// TIA Portal V19 export
VAR_GLOBAL   // PLC tag table "Safety_IO"
   IS_ZAxisBrakeFeedback AT %I500.0 : Bool;   // Robot Z axis brake status feedback channel 1   {ExternalAccessible false}
   IS_ZAxisBrakeFeedback_Ch2 AT %I500.4 : Bool;   // Robot Z axis brake status feedback channel 2   {ExternalAccessible false}
   OS_OpenZAxisBrake AT %Q508.0 : Bool;   // Open Z axis brake   {ExternalAccessible false}
   ISS_OpenZAxisBrake AT %I508.0 : Bool;   // State Open Z axis brake   {ExternalAccessible false}
   ISS_ZAxisBrakeFeedback AT %I501.0 : Bool;   // State Robot Z axis brake status feedback channel 1   {ExternalAccessible false}
   ISS_ZAxisBrakeFeedback_Ch2 AT %I501.4 : Bool;   // State Robot Z axis brake status feedback channel 2   {ExternalAccessible false}
   IS_AutomaticMode AT %I514.0 : Bool;   // True if Automatic mode is selected.   {ExternalAccessible false}
   IS_DriveEnableFeedback AT %I514.1 : Bool;   // True if the power to the motors is enabled.   {ExternalAccessible false}
   IS_EnableSwitch AT %I514.2 : Bool;   // True when the enable switch is activated   {ExternalAccessible false}
   IS_LocalEStopStatus AT %I514.3 : Bool;   // False if the emergency stop on the FlexPendant is pressed.   {ExternalAccessible false}
   IS_ManualFullSpeedMode AT %I514.4 : Bool;   // True if manual full speed mode is selected.   {ExternalAccessible false}
   IS_ManualMode AT %I514.5 : Bool;   // True if manual mode is selected.   {ExternalAccessible false}
   OS_SafetyEnable AT %Q526.1 : Bool;   // True as soon as communication is up   {ExternalAccessible false}
   IS_Stop0Status AT %I514.6 : Bool;   // False if a stop category 0 is active.   {ExternalAccessible false}
   IS_Stop1Status AT %I514.7 : Bool;   // False if a stop category 1 is active.   {ExternalAccessible false}
   OS_ExternalEStop AT %Q527.0 : Bool;   // Write external emergency stop to robot safemove   {ExternalAccessible false}
   OS_ExternalOProtect AT %Q527.1 : Bool;   // Write external operator protection to robot safemove   {ExternalAccessible false}
   IS_FdbExternalEstop AT %I515.0 : Bool;   // Feedback from robot safemove for external emergency stop   {ExternalAccessible false}
   IS_FdbExternalOProtect AT %I515.1 : Bool;   // Feedback from robot safemove for external operator protection   {ExternalAccessible false}
   ISB_Safety500 AT %IB500 : Byte;   //    {ExternalAccessible false}
   OSB_Safety508 AT %QB508 : Byte;   //    {ExternalAccessible false}
   OS_PowerOffFerRo AT %Q508.1 : Bool;   // Power Off 24v safety of FerRobotic   {ExternalAccessible false}
   ISS_PowerOffFerRo AT %I508.1 : Bool;   // State Power Off 24v safety of FerRobotic   {ExternalAccessible false}
END_VAR
